ABB RobotStudio station: RoboJengaSolution.rsstn

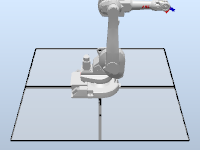
Station RoboJengaSolution (saved by RobotStudio 7.0.8666.559)
Controller IRB_1600_10kg_1.45m
  mechanical unit ROB_1: IRB1600_10_145__01, 6 joints, base frame (0, 0, 0) mm
Layout (positions relative to the parent item):
  - IRB1600_10_145__01 [mechanism, from Robots\IRB1600_10_145_G_01.rslib] at (0, 0, 0) mm; joint values [0, 0, 0, 0, 0.5236, 0] (rad or m)
